FUNCTION_BLOCK FB_PartBuild
VAR_INPUT
	iLastExpectedOP:UINT;
	iNumAttemptedRejects:UINT;
	iPartPresent: BOOL;
	iPartReadOK: BOOL;
	iPartReadNOK: BOOL;



	iStationData:typeStationMode;
	
END_VAR
VAR_OUTPUT
	qMsgNoPartRead: BOOL; //message for no part data read yet
	qMsgPartNOKBuild: BOOL; //message for part data NOK to build


END_VAR
VAR
	tDataRead: BOOL;
	retvall: UDINT;
	tserialLen: INT;
	tDescripLen: INT;
END_VAR

VAR_IN_OUT
	iqData :typeStationTask;
END_VAR
VAR // added by the converter: edge detectors and wires of the graphical bodies
    _ft1 : F_TRIG;
END_VAR

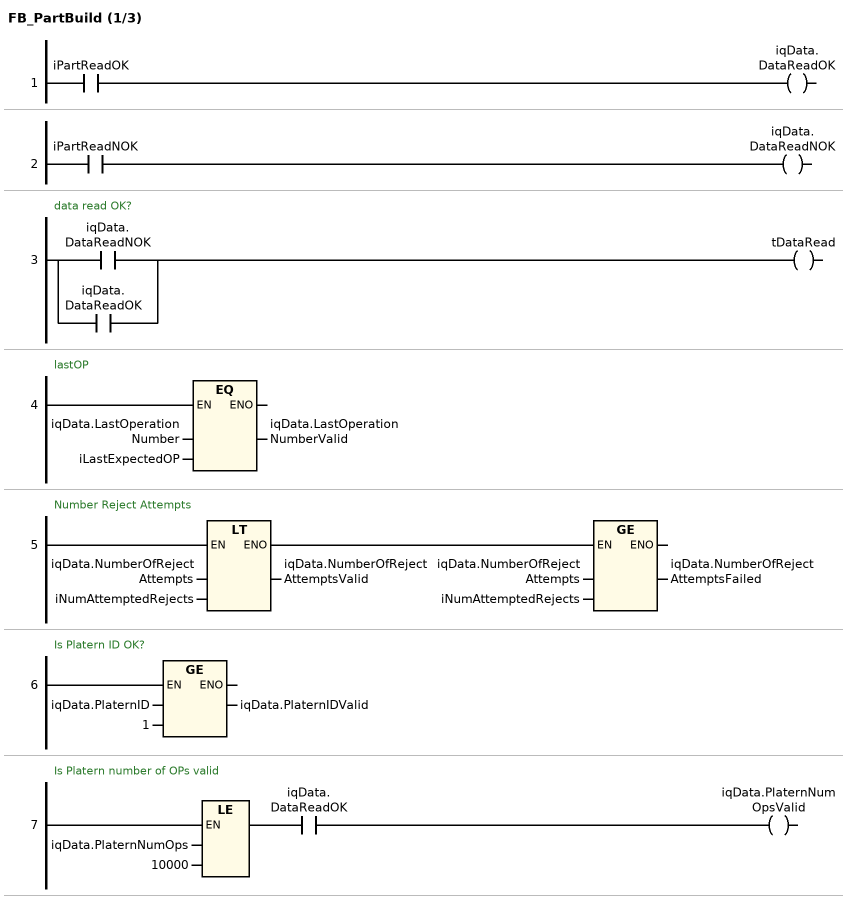
// NETWORK 1
iqData.DataReadOK := iPartReadOK;

// NETWORK 2
iqData.DataReadNOK := iPartReadNOK;

// NETWORK 3
// data read OK?
tDataRead := iqData.DataReadNOK OR iqData.DataReadOK;

// NETWORK 4
// lastOP
iqData.LastOperationNumberValid := iqData.LastOperationNumber = iLastExpectedOP;

// NETWORK 5
// Number Reject Attempts
iqData.NumberOfRejectAttemptsValid := iqData.NumberOfRejectAttempts < iNumAttemptedRejects;
iqData.NumberOfRejectAttemptsFailed := iqData.NumberOfRejectAttempts >= iNumAttemptedRejects;

// NETWORK 6
// Is Platern ID OK?
iqData.PlaternIDValid := iqData.PlaternID >= 1;

// NETWORK 7
// Is Platern number of OPs valid
iqData.PlaternNumOpsValid := iqData.PlaternNumOps <= 10000 AND iqData.DataReadOK;

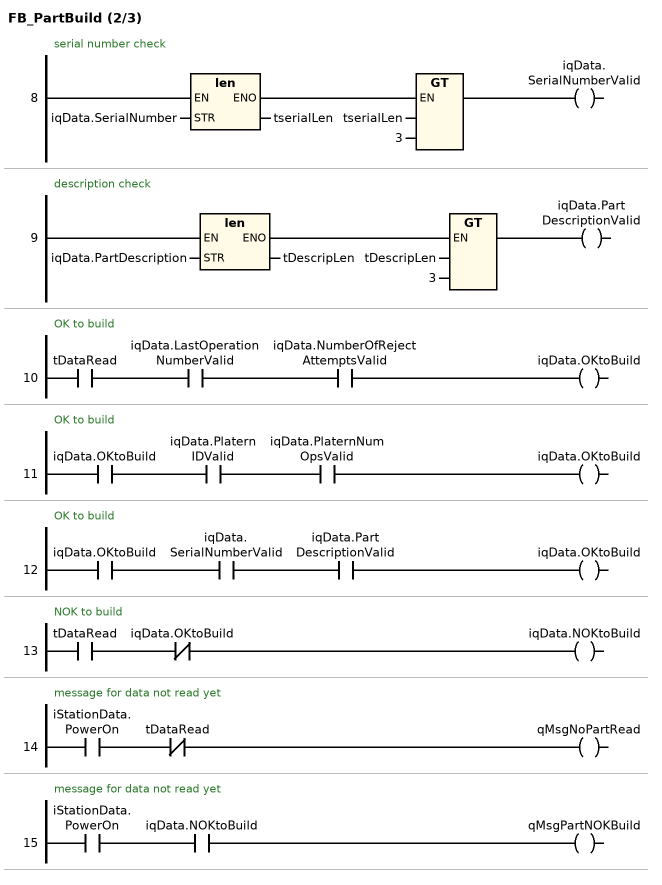
// NETWORK 8
// serial number check
tserialLen := len(STR := iqData.SerialNumber);
iqData.SerialNumberValid := tserialLen > 3;

// NETWORK 9
// description check
tDescripLen := len(STR := iqData.PartDescription);
iqData.PartDescriptionValid := tDescripLen > 3;

// NETWORK 10
// OK to build
iqData.OKtoBuild := tDataRead AND iqData.LastOperationNumberValid AND iqData.NumberOfRejectAttemptsValid;

// NETWORK 11
// OK to build
iqData.OKtoBuild := iqData.OKtoBuild AND iqData.PlaternIDValid AND iqData.PlaternNumOpsValid;

// NETWORK 12
// OK to build
iqData.OKtoBuild := iqData.OKtoBuild AND iqData.SerialNumberValid AND iqData.PartDescriptionValid;

// NETWORK 13
// NOK to build
iqData.NOKtoBuild := tDataRead AND NOT iqData.OKtoBuild;

// NETWORK 14
// message for data not read yet
qMsgNoPartRead := iStationData.PowerOn AND NOT tDataRead;

// NETWORK 15
// message for data not read yet
qMsgPartNOKBuild := iStationData.PowerOn AND iqData.NOKtoBuild;

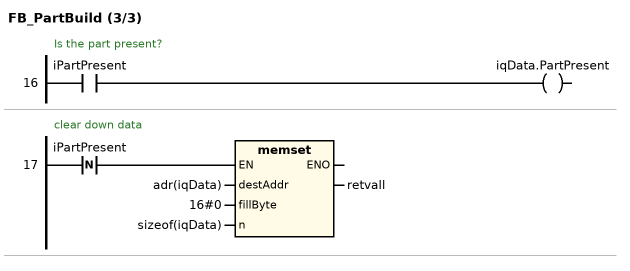
// NETWORK 16
// Is the part present?
iqData.PartPresent := iPartPresent;

// NETWORK 17
// clear down data
_ft1(CLK := iPartPresent);
IF _ft1.Q THEN retvall := memset(destAddr := adr(iqData), fillByte := 16#0, n := sizeof(iqData)); END_IF

END_FUNCTION_BLOCK

(* stored: Version 1.1.0.1, ProductVersion 3.1.4024.12
   POU FB_PartBuild: Id {bfc14baa-066e-4804-8b32-5d911ebfa702}, SpecialFunc None *)
